        // ===========================================
        // STEP 133: StoperRelease_4
        // ===========================================
        STEP_ST10_Flow26_JMagnetLoad_Unload_StoperRelease_4:
            // Action Qualifier=R
            // Token: "ST10Cylinder".Cy[36].Inout.AutoGoHome
            "ST10Cylinder".Cy[36].Inout.AutoGoHome := FALSE;
            // Action Qualifier=S
            // Token: "ST10Cylinder".Cy[36].Inout.AutoGoWork
            "ST10Cylinder".Cy[36].Inout.AutoGoWork := TRUE;

            // Transition to next step: 168
            IF TRUE THEN  // Sequential transition - review XML for actual condition
                #State := STEP_ST10_Flow26_JMagnetLoad_Unload_AriveTimeDelay_10;
            END_IF;

        // ===========================================
        // STEP 168: AriveTimeDelay_10
        // ===========================================
        STEP_ST10_Flow26_JMagnetLoad_Unload_AriveTimeDelay_10:
            // No actions in XML

            // Transition to next step: 145
            IF TRUE THEN  // Sequential transition - review XML for actual condition
                #State := STEP_ST10_Flow26_JMagnetLoad_Unload_StoperRelease_6;
            END_IF;

        // ===========================================
        // STEP 145: StoperRelease_6
        // ===========================================
        STEP_ST10_Flow26_JMagnetLoad_Unload_StoperRelease_6:
            // Action Qualifier=R
            // Token: "ST10Cylinder".Cy[38].Inout.AutoGoHome
            "ST10Cylinder".Cy[38].Inout.AutoGoHome := FALSE;
            // Action Qualifier=S
            // Token: "ST10Cylinder".Cy[38].Inout.AutoGoWork
            "ST10Cylinder".Cy[38].Inout.AutoGoWork := TRUE;

            // Transition to next step: 147
            IF TRUE THEN  // Sequential transition - review XML for actual condition
                #State := STEP_ST10_Flow26_JMagnetLoad_Unload_TimeDelay_4;
            END_IF;

        // ===========================================
        // STEP 147: TimeDelay_4
        // ===========================================
        STEP_ST10_Flow26_JMagnetLoad_Unload_TimeDelay_4:
            // No actions in XML

            // Transition to next step: 173
            IF TRUE THEN  // Sequential transition - review XML for actual condition
                #State := STEP_ST10_Flow26_JMagnetLoad_Unload_AriveTimeDelay_11;
            END_IF;

        // ===========================================
        // STEP 173: AriveTimeDelay_11
        // ===========================================
        STEP_ST10_Flow26_JMagnetLoad_Unload_AriveTimeDelay_11:
            // No actions in XML

            // Transition to next step: 162
            IF TRUE THEN  // Sequential transition - review XML for actual condition
                #State := STEP_ST10_Flow26_JMagnetLoad_Unload_StoperRelease_8;
            END_IF;

        // ===========================================
        // STEP 162: StoperRelease_8
        // ===========================================
        STEP_ST10_Flow26_JMagnetLoad_Unload_StoperRelease_8:
            // Action Qualifier=R
            // Token: "ST10Cylinder".Cy[33].Inout.AutoGoHome
            "ST10Cylinder".Cy[33].Inout.AutoGoHome := FALSE;
            // Action Qualifier=S
            // Token: "ST10Cylinder".Cy[33].Inout.AutoGoWork
            "ST10Cylinder".Cy[33].Inout.AutoGoWork := TRUE;

            // Transition to next step: 42
            IF TRUE THEN  // Sequential transition - review XML for actual condition
                #State := STEP_ST10_Flow26_JMagnetLoad_Unload_WaitLineMotorReady_2;
            END_IF;

        // ===========================================
        // STEP 42: WaitLineMotorReady_2
        // ===========================================
        STEP_ST10_Flow26_JMagnetLoad_Unload_WaitLineMotorReady_2:
            // No actions in XML

            // Transition to next step: 48
            IF TRUE THEN  // Sequential transition - review XML for actual condition
                #State := STEP_ST10_Flow26_JMagnetLoad_Unload_WaitPalletArrveNextPos_3;
            END_IF;

        // ===========================================
        // STEP 48: WaitPalletArrveNextPos_3
        // ===========================================
        STEP_ST10_Flow26_JMagnetLoad_Unload_WaitPalletArrveNextPos_3:
            // Action Qualifier=S
            // Token: "MotorControl".Dev[13].Auto.Start
            "MotorControl".Dev[13].Auto.Start := TRUE;
            // Action Qualifier=R
            // Token: "MotorControl".Dev[13].Auto.CCWStart
            "MotorControl".Dev[13].Auto.CCWStart := FALSE;
            // Action Qualifier=R
            // Token: "MotorControl".Dev[2].Auto.CCWStart
            "MotorControl".Dev[2].Auto.CCWStart := FALSE;
            // Action Qualifier=S
            // Token: "MotorControl".Dev[2].Auto.Start
            "MotorControl".Dev[2].Auto.Start := TRUE;

            // Transition to next step: 65
            IF TRUE THEN  // Sequential transition - review XML for actual condition
                #State := STEP_ST10_Flow26_JMagnetLoad_Unload_WaitLineMotorReady_7;
            END_IF;

        // ===========================================
        // STEP 65: WaitLineMotorReady_7
        // ===========================================
        STEP_ST10_Flow26_JMagnetLoad_Unload_WaitLineMotorReady_7:
            // No actions in XML

            // Transition to next step: 130
            IF TRUE THEN  // Sequential transition - review XML for actual condition
                #State := STEP_ST10_Flow26_JMagnetLoad_Unload_AriveTimeDelay_4;
            END_IF;

        // ===========================================
        // STEP 130: AriveTimeDelay_4
        // ===========================================
        STEP_ST10_Flow26_JMagnetLoad_Unload_AriveTimeDelay_4:
            // No actions in XML

            // Transition to next step: 124
            IF TRUE THEN  // Sequential transition - review XML for actual condition
                #State := STEP_ST10_Flow26_JMagnetLoad_Unload_TimeDelay;
            END_IF;

        // ===========================================
        // STEP 124: TimeDelay
        // ===========================================
        STEP_ST10_Flow26_JMagnetLoad_Unload_TimeDelay:
            // No actions in XML

            // Transition to next step: 2
            IF TRUE THEN  // Sequential transition - review XML for actual condition
                #State := STEP_ST10_Flow26_JMagnetLoad_Unload_S2;
            END_IF;

        // ===========================================
        // STEP 2: S2
        // ===========================================
        STEP_ST10_Flow26_JMagnetLoad_Unload_S2:
            // No actions in XML

            // Transition to next step: 241
            IF TRUE THEN  // Sequential transition - review XML for actual condition
                #State := STEP_ST10_Flow26_JMagnetLoad_Unload_Process_Finish_5;
            END_IF;

        // ===========================================
        // STEP 241: Process Finish_5
        // ===========================================
        STEP_ST10_Flow26_JMagnetLoad_Unload_Process_Finish_5:
            // No actions in XML

            // Transition to next step: 139
            IF TRUE THEN  // Sequential transition - review XML for actual condition
                #State := STEP_ST10_Flow26_JMagnetLoad_Unload_WaitPalletArive_3;
            END_IF;

        // ===========================================
        // STEP 139: WaitPalletArive_3
        // ===========================================
        STEP_ST10_Flow26_JMagnetLoad_Unload_WaitPalletArive_3:
            // Action Qualifier=N
            // Token: "AutoProcessControl".Global.J.EmptyStopRequestPallet_1
            "AutoProcessControl".Global.J.EmptyStopRequestPallet_1;

            // Transition to next step: 240
            IF TRUE THEN  // Sequential transition - review XML for actual condition
                #State := STEP_ST10_Flow26_JMagnetLoad_Unload_Process_Finish_4;
            END_IF;

        // ===========================================
        // STEP 240: Process Finish_4
        // ===========================================
        STEP_ST10_Flow26_JMagnetLoad_Unload_Process_Finish_4:
            // No actions in XML

    END_CASE;

    // UPDATE ioPM_Inface
    #ioPM_Inface.InitialRun := #act_InitialRun;
    #ioPM_Inface.InitialOK := #act_InitialOK;
    #ioPM_Inface.WaitRunning := #act_WaitRunning;
    #ioPM_Inface.Running := #act_Running;
    #ioPM_Inface.ProcessComplete := #act_ProcessComplete;
    #ioPM_Inface.ProcessStart := #act_ProcessStart;
    #ioPM_Inface.UnPause := #act_UnPause;

    // ERROR HANDLING
    IF #bError THEN
        #ioStatus := 900;
        #oAlarmID := INT_TO_WORD(#wErrorID);
    ELSE
        #ioStatus := 0;
        #oAlarmID := 0;
    END_IF;
END_FUNCTION_BLOCK

//=============================================================================
// END OF FILE
//=============================================================================
